# EPICS StreamDevice protocol: EPICS/rek.proto
# Author: Philip Weigel

Terminator = CR;

# Voltage (Hex)
set_voltage {
    out "#\$1 CH0 %04X";
}

get_voltage {
    out "#\$1 CH0?";
    in "CH0=%XH"
}

read_voltage {
    out "#\$1 MN1";
    in "MONI1=%XH";
}

# Current (Hex)
set_current {
    out "#\$1 CH1 %04X";
}

get_current {
    out "#\$1 CH1?";
    in "CH1=%XH"
}

read_current {
    out "#\$1 MN2";
    in "MONI2=%XH";
}

# Status
reset {
    out "#\$1 REN";
    #out "#\$1 RST";
}

enable_output {
    out "#\$1 REN";
	out "#\$1 ICN 100";
	out "#\$1 SW1";
}

disable_output {
	out "#\$1 SW0";
}

set_status {
    out "#\$1 SW%d";

    @init {
      reset;
    }
}

read_status {
    out "#\$1 STS";

    in "#%*d %{CF|CO} %*c%*c %*c%*c";
}
